FUNCTION_BLOCK fbSlidingDoorCtrl
VAR_INPUT

	bEnable				: BOOL;
	bEmergencyStop		: BOOL;
	bDoorOpenExe		: BOOL;
	bDoorCloseExe		: BOOL;
	bDoorOpenRS		: BOOL;
	bDoorCloseRS		: BOOL;
	bDoorUnlockRS		: BOOL;
	bDoorUnclampRS		: BOOL;
	bLowVacuumSignal	: BOOL;

END_VAR
VAR_OUTPUT

	bDoorOpenOutPut			: BOOL;
	bDoorCloseOutPut		: BOOL;
	bDoorOpenCompleted		: BOOL;
	bDoorCloseCompleted		: BOOL;
	bDoorUnlockOutPut		: BOOL;
	bDoorUnclampOutPut		: BOOL;
	bVacuumReleaseValve	: BOOL;

END_VAR



VAR
	step1:BOOL;
	step2:BOOL;
	step3:BOOL;
	step4:BOOL;
	step5:BOOL;
	step6:BOOL;


END_VAR

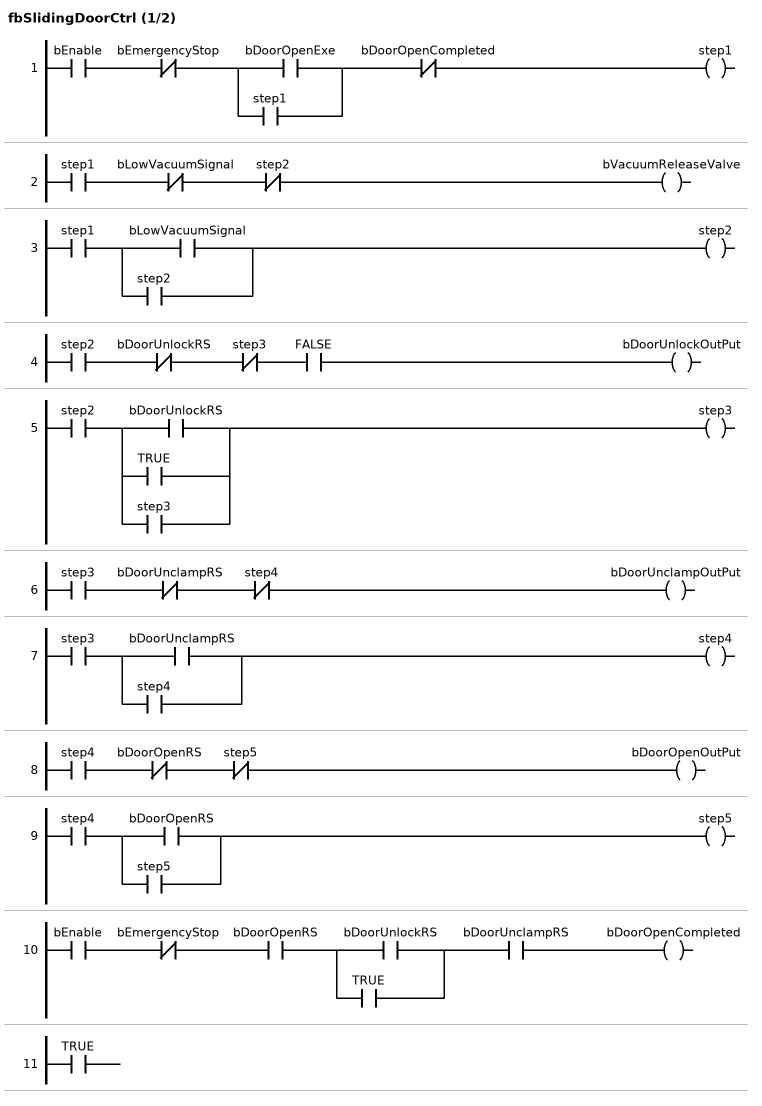
// NETWORK 1
step1 := (bEnable AND NOT bEmergencyStop AND (bDoorOpenExe OR step1)) AND NOT bDoorOpenCompleted;

// NETWORK 2
bVacuumReleaseValve := step1 AND NOT bLowVacuumSignal AND NOT step2;

// NETWORK 3
step2 := step1 AND (bLowVacuumSignal OR step2);

// NETWORK 4
bDoorUnlockOutPut := step2 AND NOT bDoorUnlockRS AND NOT step3 AND FALSE;

// NETWORK 5
step3 := step2 AND (bDoorUnlockRS OR TRUE OR step3);

// NETWORK 6
bDoorUnclampOutPut := step3 AND NOT bDoorUnclampRS AND NOT step4;

// NETWORK 7
step4 := step3 AND (bDoorUnclampRS OR step4);

// NETWORK 8
bDoorOpenOutPut := step4 AND NOT bDoorOpenRS AND NOT step5;

// NETWORK 9
step5 := step4 AND (bDoorOpenRS OR step5);

// NETWORK 10
bDoorOpenCompleted := (bEnable AND NOT bEmergencyStop AND bDoorOpenRS AND (bDoorUnlockRS OR TRUE)) AND bDoorUnclampRS;

// NETWORK 11

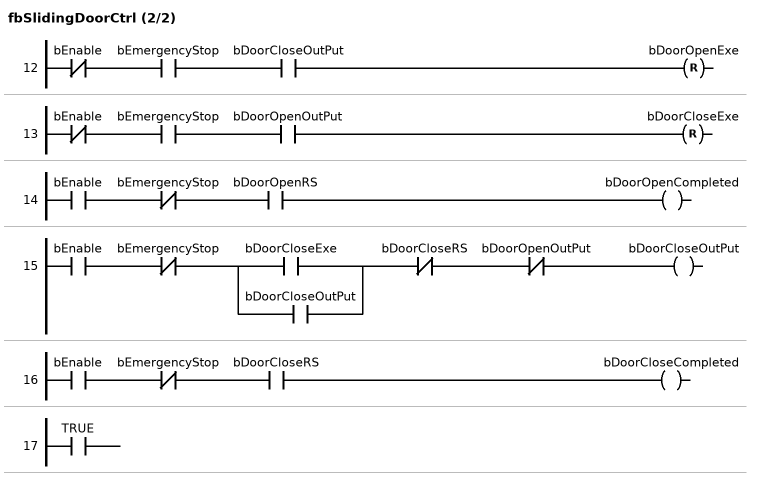
// NETWORK 12
bDoorOpenExe R= NOT bEnable AND bEmergencyStop AND bDoorCloseOutPut;

// NETWORK 13
bDoorCloseExe R= NOT bEnable AND bEmergencyStop AND bDoorOpenOutPut;

// NETWORK 14
bDoorOpenCompleted := bEnable AND NOT bEmergencyStop AND bDoorOpenRS;

// NETWORK 15
bDoorCloseOutPut := (bEnable AND NOT bEmergencyStop AND (bDoorCloseExe OR bDoorCloseOutPut)) AND NOT bDoorCloseRS AND NOT bDoorOpenOutPut;

// NETWORK 16
bDoorCloseCompleted := bEnable AND NOT bEmergencyStop AND bDoorCloseRS;

// NETWORK 17

END_FUNCTION_BLOCK

(* stored: Version 1.1.0.1, ProductVersion 3.1.4024.12
   POU fbSlidingDoorCtrl: Id {0a19330c-6fe0-406c-9d3f-1c3e9d5bd86d}, SpecialFunc None *)
